PROGRAM MAIN
VAR
    rTrig_BP_EG  : R_TRIG;
    rTrig_BP_1OG : R_TRIG;
    rTrig_BP_2OG : R_TRIG;
END_VAR

rTrig_BP_EG(CLK := GVL.BP_EG);
rTrig_BP_1OG(CLK := GVL.BP_1OG);
rTrig_BP_2OG(CLK := GVL.BP_2OG);

// Appelle bouton etage
IF rTrig_BP_EG.Q THEN
	GVL.iEtageAppel := 0;
	gvl.MouvementAscenseur := TRUE;
END_IF

IF rTrig_BP_1OG.Q THEN
	GVL.iEtageAppel := 1;
	gvl.MouvementAscenseur := TRUE;
END_IF

IF rTrig_BP_2OG.Q THEN
	GVL.iEtageAppel := 2;
	gvl.MouvementAscenseur := TRUE;
END_IF

// Fermeture porte
IF gvl.MouvementAscenseur THEN
	gvl.FermeturePorte (In := TRUE, PT :=  T#5S);
END_IF

// Durée du trajet
IF gvl.FermeturePorte.Q THEN
	
	// Lampe Fermeture
	gvl.Lampe_Fermeture := TRUE;	
	gvl.Lampe_Ouverture := False;

	// Lampe témoin chaque étage
	gvl.Lampe_EG := FALSE;
	gvl.Lampe_1OG := FALSE;
	gvl.Lampe_2OG := false;
	
	// Calcul du temps
	CASE ABS(GVL.iEtageAppel - GVL.iEtageActuel) OF

        0: GVL.TempsMouvementAscenseur (IN := TRUE, PT := T#0S);
        1: GVL.TempsMouvementAscenseur (IN := TRUE, PT := T#5S);
        2: GVL.TempsMouvementAscenseur (IN := TRUE, PT := T#10S);
		
    END_CASE
	
	// Arrivé a l'étage demandé
	IF GVL.TempsMouvementAscenseur.Q THEN
        GVL.iEtageActuel := GVL.iEtageAppel;
        gvl.MouvementAscenseur := FALSE;
        GVL.TempsMouvementAscenseur(IN := FALSE);
		
		CASE GVL.iEtageActuel OF
			0:
				GVL.BP_EG := FALSE;
				GVL.Lampe_EG := TRUE;
		
			1:
				GVL.BP_1OG := FALSE;
				GVL.Lampe_1OG := TRUE;
		
			2:
				GVL.BP_2OG := FALSE;
				GVL.Lampe_2OG := TRUE;
		END_CASE
		
		gvl.Lampe_Fermeture := FALSE;
		
		// Ouverture porte
		gvl.OuverturePorte (In := TRUE, PT :=  T#5S);
		
		IF gvl.OuverturePorte.Q THEN
			gvl.Lampe_Ouverture := TRUE;
		END_IF
    END_IF
END_IF

END_PROGRAM

(* stored: Version 1.1.0.1, ProductVersion 3.1.4024.16
   POU MAIN: Id {3f45254e-648f-4ffc-a0fd-e9e2d67bcb4f}, SpecialFunc None *)
